FUNCTION_BLOCK GernericErrorWatchdog_t  
VAR_INPUT
END_VAR
VAR_OUTPUT
END_VAR
VAR
	_alarm : FB_TcAlarm; 	// the alarm object
	_init : BOOL := FALSE;  // if true the object is initialised
	_timer : TON; 			// counts the time
	_sensor : BOOL; 		// if true reset timer
	_isAlarmDisplayed : BOOL := FALSE; // if true, the alarm wasn't deleted from the event logger 
	_isAlarmClearedLast : BOOL := FALSE; // true when the alarm has been cleard last
	_waitHWConformation : BOOL := TRUE; // if true, the watchdogs wait for the correct value bevore clearing the error.
	
	_eventLogger : FB_TcEventLogger;
	_eventLoggerSettings : FB_TcClearLoggedEventsSettings;
	_eventLoggerFilter : FB_TcEventFilter;
END_VAR

// confirm the alarm
METHOD confirm : BOOL
VAR_INPUT
END_VAR
IF _init = FALSE THEN
	confirm := FALSE; 
	RETURN;
END_IF

_alarm.Confirm();

// restet timeout
_timer.IN := FALSE;
_timer();

confirm := TRUE;
END_METHOD

// returns true if the alarm is raised
METHOD isAlarmRaised : BOOL
VAR_INPUT
END_VAR
IF _init = FALSE THEN
	isAlarmRaised := FALSE;
	return;
END_IF

isAlarmRaised := _alarm.bActive;
RETURN;
END_METHOD

// registers a error state or reregister an existing error state
METHOD register : bool
VAR_INPUT
	stEventEntity : TcEventEntry;
	timerTime : TIME; // sets the timer for the timeout
	conformation : BOOL := TRUE; 
	waitHWConformation : bool := TRUE;
END_VAR
_alarm.CreateEx(stEventEntity, conformation);
_timer.PT := timerTime;
_init := TRUE;
_waitHWConformation := waitHWConformation; 
RETURN;
END_METHOD

// resets the alarm. Only use this as a last resort.
METHOD reset : BOOL
VAR_INPUT
END_VAR
IF _init = FALSE THEN
	reset := FALSE;
	RETURN;
END_IF

_alarm.Confirm();
_alarm.Clear(bResetConfirmation := TRUE);

_timer.IN := FALSE;
_timer(); 

reset := TRUE;
RETURN;
END_METHOD

// call this function every cycle. 
METHOD update : bool
VAR_INPUT
	sensor : bool; // if true the sensor is active and the watchdog resets, if it isn't set, the time starts.
END_VAR
IF _init = FALSE THEN
	update := FALSE; 
	RETURN;
END_IF



IF sensor = FALSE THEN
	_timer.IN := TRUE;
ELSE 
	_timer.IN := FALSE;
END_IF

_timer();

// clear alarm from log
IF (_alarm.bActive = FALSE AND _isAlarmDisplayed) OR _isAlarmClearedLast THEN
	_isAlarmDisplayed := FALSE;
	_isAlarmClearedLast := FALSE;
	_eventLoggerFilter.EventClass.EqualTo(value := _alarm.EventClass);
	_eventLoggerSettings.AddFilter(_eventLoggerFilter);
	_eventLogger.ClearLoggedEvents(_eventLoggerSettings);
	_eventLogger.ClearLoggedEvents(_eventLoggerSettings);
END_IF

IF _timer.Q AND _alarm.bActive = FALSE THEN
	// timeout detected
	_alarm.Raise(); 
	_isAlarmDisplayed := TRUE; 
END_IF

IF _alarm.bRaised AND (sensor OR _waitHWConformation = FALSE) THEN
	_alarm.Clear();
	_isAlarmClearedLast := NOT _alarm.bActive;
END_IF

update := TRUE;
RETURN;
END_METHOD

END_FUNCTION_BLOCK

(* stored: Version 1.1.0.1
   POU GernericErrorWatchdog_t: Id {f3f41f7b-8e73-4739-bc75-658a23f6a753}, SpecialFunc None
   Method confirm: Id {7074bfe5-b899-469f-bbf3-e3147b59627b}
   Method isAlarmRaised: Id {9a2b46c8-5918-4beb-bab5-0fcdb4329d16}
   Method register: Id {d8f783b0-24d7-4051-b052-66edd70897cb}
   Method reset: Id {1ad239a2-4e66-4c00-8dad-45c8d1b4fdb7}
   Method update: Id {3366293f-fa44-4d2c-9b3d-cd3a48dd9804} *)
